Staubli VAL3: ISOConnect.pgx

program ISOConnect()
  local num l_nLength
begin

  nISO_CR[16]=nLocalTSAP_HI
  nISO_CR[17]=nLocalTSAP_LO
  nISO_CR[20]=nRemoteTSAP_HI
  nISO_CR[21]=nRemoteTSAP_LO

  //if sioSet(sTCPclient, nISO_CR) == size(nISO_CR)
  call sendPacket(nISO_CR, size(nISO_CR))
  if nLastError==nNoErrors
    call recvISOpacket(l_nLength)
    //15 = 22 (sizeof CC telegram) - 7 (sizeof Header)
    if nLastError==nNoErrors and l_nLength==15
      //it was a connection confirm?
      if nLastPDUType!=nCC
        call setLastError(nErrISOInvPDU)
      endIf
    endIf
  else
    call setLastError(nErrISOConnFail)
  endIf

end
